// TIA Portal V17 export
// export: Created 2025-03-11T12:28:51.3304256Z, ExportSetting WithDefaults, DisplayName Totally Integrated Automation Portal, DisplayVersion V17 Update 8, DisplayName TIA Portal Openness, DisplayVersion V17 Update 8, DisplayName TIA Portal Version Control Interface, DisplayVersion V17, DisplayName SINAMICS Startdrive Advanced, DisplayVersion V17 SP2, DisplayName SINAMICS Startdrive G110M, G120, G120C, G120D, G120P, G115D, DisplayVersion V17 SP2, DisplayName SINAMICS Startdrive G130, G150, S120, S150, SINAMICS MV, S210, DisplayVersion V17 SP2, DisplayName STEP 7 Professional, DisplayVersion V17 Update 8, DisplayName SINUMERIK ONE STEP 7 Toolbox, DisplayVersion V17 Update 12, DisplayName SINUMERIK 840D sl STEP 7 Toolbox, DisplayVersion V17 Update 12, DisplayName STEP 7 Safety, DisplayVersion V17 Update 6, DisplayName WinCC Advanced, DisplayVersion V17 Update 8
DATA_BLOCK "DB21223_POWDER_SEQUENCES_COORDINATOR"   // DB21223
{ S7_Optimized_Access := 'FALSE'; DB_Accessible_From_OPC_UA := 'FALSE' }
VERSION : 0.1
// stored: AutoNumber false, DBAccessibleFromOPCUA false, DBAccessibleFromWebserver true, IsOnlyStoredInLoadMemory false, IsWriteProtectedInAS false
   VAR
      UNIT_01_POWDER_FEEDER_1_LINE_1 : Struct
         HMI_HIGH_CURRENT_LIMIT : Real;   // UNIT 01 POWDER FEEDER 1 LINE 1 HMI HIGH CURRENT LIMIT
         HMI_LOW_CURRENT_LIMIT : Real;   // HMI LOW CURRENT LIMIT
         POWDER_FILLING_STOP_BY_CURRENT : Bool;   // UNIT 01 POWDER FEEDER 1 LINE 1 POWDER FILLING STOP BY CURRENT
         "POWDER_FILLING_START_BY CURRENT" : Bool;   // UNIT 01 POWDER FEEDER 1 LINE 1 POWDER FILLING START BY CURRENT
      END_STRUCT;
      UNIT_01_POWDER_FEEDER_1_LINE_2 : Struct
         HMI_HIGH_CURRENT_LIMIT : Real;   // HMI HIGH CURRENT LIMIT
         HMI_LOW_CURRENT_LIMIT : Real;   // HMI LOW CURRENT LIMIT
         POWDER_FILLING_STOP_BY_CURRENT : Bool;   // UNIT 01 POWDER FEEDER 1 LINE 2 POWDER FILLING STOP BY CURRENT
         "POWDER_FILLING_START_BY CURRENT" : Bool;   // UNIT 01 POWDER FEEDER 1 LINE 2 POWDER FILLING START BY CURRENT
      END_STRUCT;
   END_VAR
BEGIN
END_DATA_BLOCK
